# EPICS substitutions: modules/event/evrSupport/Db/ioc/IOC-IN20-PM07evr.substitutions
#==============================================================================
#
# Abs:  LCLS EVR IOC records for IN20 PM07
#
# Name: IOC-IN20-PM07evr.substitutions
#
#==============================================================================
#
file evrPMXX.db
{
pattern { DEVICE        }
	{ EVR:IN20:PM07 }
}
